// TIA Portal V19 export
FUNCTION_BLOCK "RPM_to_MPM"   // FB22, LAD
{ S7_Optimized_Access := 'TRUE' }
// stored: AutoNumber false, MemoryReserve 100, SetENOAutomatically false
   VAR_INPUT
      RPM : LReal;
      Diameter : LReal;
   END_VAR
   VAR_OUTPUT
      MRM : Int;   // Input for HMI gauge
   END_VAR
BEGIN

REGION Network 1: Rev Per Minute to Meters Per Minute MRM = (RPM * Diameter) * Pi
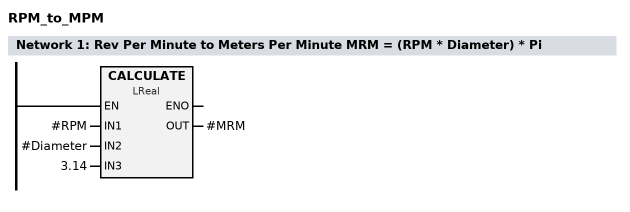
   RUNG wire#powerrail
      { S7_Templates := "SrcType := LReal"; S7_Expression := "(IN2*IN3)*IN1" } Calculate(in1 := #RPM, in2 := #Diameter, in3 := 3.14, out => #MRM)
   END_RUNG
   // the same network as SCL:
   #MRM := (#Diameter*3.14)*#RPM;
END_REGION
END_FUNCTION_BLOCK
